// Mitsubishi GX Works2 project: 2   PLC: FX3U/FX3UC

// task Task_01 (event TRUE, interval 0, priority 31): POU_01

PROGRAM POU_01
VAR
  wstep : INT;
END_VAR
IF M8002 THEN
	wstep := 0;
END_IF;

IF M3 THEN
	wstep := 90;
END_IF;

CASE wstep OF
	0:
	Y3 := TRUE;
	Y0 := FALSE;
	Y1 := FALSE;
	
	IF M1 THEN
		wstep := 20;
	END_IF;
	
	IF M2 THEN
		wstep := 30;
	END_IF;
	
	20:
	Y0 := TRUE;
	Y3 := FALSE;
	IF M0 THEN
		wstep := 0;
	END_IF;
	
	30:
	Y1 := TRUE;
	Y3 := FALSE;
	IF M0 THEN
		wstep := 0;
	END_IF;
	
	90:
	Y2 := TRUE;
	Y3 := TRUE;
	Y0 := FALSE;
	Y1 := FALSE;
	
	IF NOT M3 THEN
		wstep := 0;
	END_IF;
END_CASE;
END_PROGRAM
